{attribute 'qualified_only'}
{attribute 'strict'}
TYPE ServerityLevelType :
(
	SERVICE := 0,
	ERROR,
	WARNING,
	INFO,
	DEBUG
);
END_TYPE

(* stored: Version 1.1.0.1, ProductVersion 3.1.4024.12
   DUT ServerityLevelType: Id {e98dd4df-9e6b-4a92-bc89-043454643b78} *)
